Omron CX-Programmer project NewProject (CX-Programmer 9.61)

# PLC NewPLC1: CP1E N30

## Global symbols (name address type ; comment)
0.00 BOOL  ; STOP
0.01 BOOL  ; START
0.02 BOOL  ; Tmbl Masuk
0.03 BOOL  ; Sensor Masuk
0.04 BOOL  ; Sensor Keluar
0.05 BOOL  ; krcs diserahkan ptgs
0.06 BOOL  ; RESET
100.00 BOOL  ; NYALA
100.01 BOOL  ; Karcis In
100.02 BOOL  ; Portal Masuk
100.03 BOOL  ; Portal Keluar
100.04 BOOL  ; Indikator Penuh
C001 BOOL  ; FULL

## Program NewProgram1 (cyclic task 0)

### Section Section1

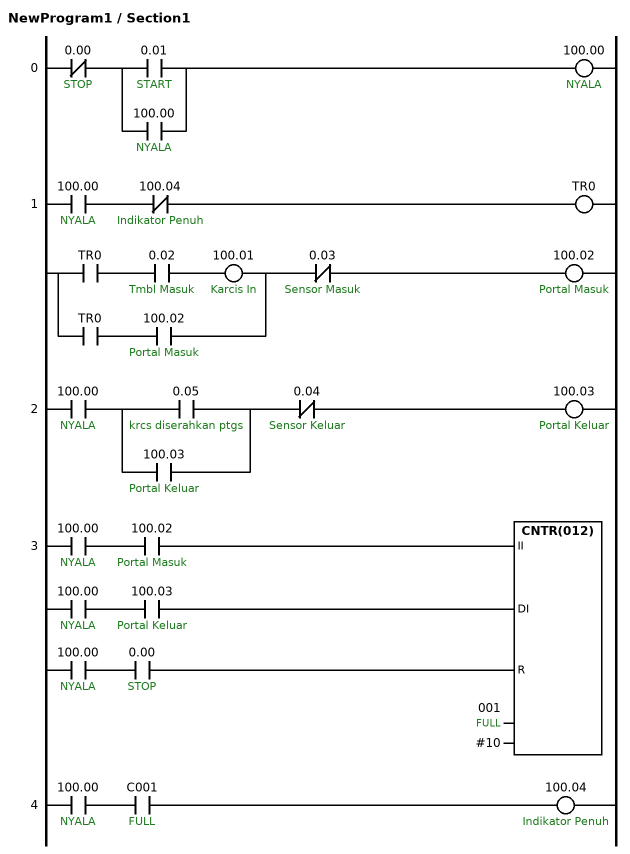
; rung 0
LDNOT 0.00  ; STOP
LD 0.01  ; START
OR 100.00  ; NYALA
ANDLD
OUT 100.00  ; NYALA
; rung 1
LD 100.00  ; NYALA
ANDNOT 100.04  ; Indikator Penuh
OUT TR0
AND 0.02  ; Tmbl Masuk
OUT 100.01  ; Karcis In
LD TR0
AND 100.02  ; Portal Masuk
ORLD
ANDNOT 0.03  ; Sensor Masuk
OUT 100.02  ; Portal Masuk
; rung 2
LD 100.00  ; NYALA
LD 0.05  ; krcs diserahkan ptgs
OR 100.03  ; Portal Keluar
ANDLD
ANDNOT 0.04  ; Sensor Keluar
OUT 100.03  ; Portal Keluar
; rung 3
LD 100.00  ; NYALA
AND 100.02  ; Portal Masuk
LD 100.00  ; NYALA
AND 100.03  ; Portal Keluar
LD 100.00  ; NYALA
AND 0.00  ; STOP
CNTR(012) 001 #10  ; FULL
; rung 4
LD 100.00  ; NYALA
AND C001  ; FULL
OUT 100.04  ; Indikator Penuh

### Section END
; rung 0
END(001)